KUKA KRL program: SCHUNK_GRASPINGKIT.src, SCHUNK_GRASPINGKIT.dat

--- SCHUNK_GRASPINGKIT.src ---
&ACCESS RVO4
&REL 37
&PARAM EDITMASK = *
&PARAM TEMPLATE = C:\KRC\Roboter\Template\ExpertVorgabe
&PARAM DISKPATH = KRC:\R1\Program\2DG
DEF SCHUNK_GRASPINGKIT( )
   INT v,s,c
   ;FOLD INI
      ;FOLD BASISTECH INI
         BAS (#INITMOV,0 )
      ;ENDFOLD (BASISTECH INI)
      ;FOLD USER INI
         ;Make your modifications here
      ;ENDFOLD (USER INI)
      ;ENDFOLD (INI)
   ;Example Program
   ;Init SVC
   SCHUNK_connect_SVC()
   v=SCHUNK_getVersion_SVC()
   ;If not v>=4 you need to update your device
   s=SCHUNK_getState_SVC()
   s=SCHUNK_getState_SVC()
   ;Add error handling if not s==2, meaning SVC is not operational
   SCHUNK_register_SVC()
   ;Init Robot and gripper
   ;Load the project that matches your application. Here project 14
   SCHUNK_setProject_SVC(14)
   ;Activate tool and workspace
   SCHUNK_setTool_SVC(1)
   SCHUNK_setWorkspace_SVC(1)
   ;Set grasp mode and object class according to your application
   SCHUNK_getGrasp_SVC(3,0,1)
   ;Different example with specified objectID=8 and graspMode=2
   ;SCHUNK_getGrasp_SVC(2,8,2)
   ;Check your edits in the $config.dat to see to which global variales the result was written
   ;Add your own error handling if replyCodeSCHUNK is not 1 meaning no part was grasped
   ;Activate your feeding system if candidateCountSCHUNK is too low
   ;Send Grasp Feedback (no effect in V4)
   SCHUNK_graspFeedback_SVC(0)
   ;Get count of all objects without planning a grasp
   c=SCHUNK_objectCount_SVC(1)
   ;with specified ObjectID
   ;c=SCHUNK_objectCount_SVC(8)
   ;Send robot pose (for robot calibration) Make sure robot position is in correct tool and base for this
   SCHUNK_robotCalib_SVC()
   ;Disconnect once finished
   SCHUNK_disconnect_SVC()
END
;FOLD SCHUNK 2D Grasping Kit Methods
   ;www.schunk.com/vision
   ;Includes methods to use the TCP/IP connection of the 2D Grasping Kit and use its commands
   ;This is not intended to move your robot, call this functions for your custom project
   ;Provided by: SCHUNK SE & Co. KG
   ;Author: Fabian Reinwald
   ;Created: 24.07.2023
   ;Last changed: 11.06.2025
   ;Keep in mind that this here needs a SCHUNK_2DGrasping.xml EthernetKRL configuration file
   ;<ETHERNETKRL>
   ;<CONFIGURATION>
      ;<EXTERNAL>
         ;<IP>172.31.1.76</IP>
         ;<PORT>42001</PORT>
         ;<TYPE>Server</TYPE>
      ;</EXTERNAL>
   ;</CONFIGURATION>
   ;<RECEIVE>
      ;<RAW>
         ;<ELEMENT Tag="SVCResponse" Type="BYTE" Set_Flag="12" SIZE="80" />
      ;</RAW>
   ;</RECEIVE>
   ;<SEND>
      ;<RAW>
         ;<ELEMENT Tag="SVCRequest" TYPE="BYTE" Set_Flag="13" SIZE="80"/>
      ;</RAW>
   ;</SEND>
   ;</ETHERNETKRL>
   ;File has to be stored at Config/User/Common/EthernetKRL/SCHUNK_2DGrasping.xml
   ;IP describes the IP adress that was set in the network settings of the SVC(SCHUNK Vision Controller)
   ;$Flag12 is used to show an incoming connection, change in xml file if needed and EKI_FLAG in .dat
   ;Tested with EthernetKRL 3.2.4
;ENDFOLD (SCHUNK 2D Grasping Kit Methods)
;Calling this function first is mandatory to establish a connection
GLOBAL DEF SCHUNK_connect_SVC()
   RET=EKI_Init("SCHUNK_2DGrasping")
   RET=EKI_Open("SCHUNK_2DGrasping")
END
;Returns the highest supported comm version by the SCHUNK Vision Controller
GLOBAL DEFFCT INT SCHUNK_getVersion_SVC()
   Prefix[]=SVC_prefix()
   Header[]=SVC_header(getVersionCode)
   Body[]=SVC_empty_body()
   OFFSET=0
   CAST_TO(Request[],OFFSET,Prefix[],Header[],Body[])
   RET = EKI_Send("SCHUNK_2DGrasping",Request[])
   FOR i=1 TO 80
      Response[i]=0
   ENDFOR
   WAIT FOR $FLAG[EKI_FLAG]
   RET=EKI_GetString("SCHUNK_2DGrasping","SVCResponse",Response[])
   $FLAG[EKI_FLAG]=FALSE
   OFFSET=10
   CAST_FROM(Response[],OFFSET,versionBuffer[])
   ;Buffers to variables
   versionSCHUNK=uint16_to_int(versionBuffer[])
   RETURN(versionSCHUNK)
ENDFCT
;Requests the current state of the SCHUNK Vision Controller.
;For state=/=2 you should probably code some exception handling as the device is not operational is that case
GLOBAL DEFFCT INT SCHUNK_getState_SVC()
   Prefix[]=SVC_prefix()
   Header[]=SVC_header(getStateCode)
   Body[]=SVC_empty_body()
   OFFSET=0
   CAST_TO(Request[],OFFSET,Prefix[],Header[],Body[])
   RET = EKI_Send("SCHUNK_2DGrasping",Request[])
   FOR i=1 TO 80
      Response[i]=0
   ENDFOR
   WAIT FOR $FLAG[EKI_FLAG]
   RET=EKI_GetString("SCHUNK_2DGrasping","SVCResponse",Response[])
   $FLAG[EKI_FLAG]=FALSE
   OFFSET=12
   CAST_FROM(Response[],OFFSET,stateBuffer[])
   stateSCHUNK=uint8_to_int(stateBuffer[])
   RETURN(stateSCHUNK)
ENDFCT
;This lets the SCHUNK Vision Controller know that it is connected to a KUKA Robot
;Calling this is the easiest way to check if your communication is working
GLOBAL DEF SCHUNK_register_SVC()
   Prefix[]=SVC_prefix()
   Header[]=SVC_header(registerClient)
   Body[]=SVC_register_client_body()
   OFFSET=0
   CAST_TO(Request[],OFFSET,Prefix[],Header[],Body[])
   RET = EKI_Send("SCHUNK_2DGrasping",Request[])
   FOR i=1 TO 80
      Response[i]=0
   ENDFOR
   WAIT FOR $FLAG[EKI_FLAG]
   RET=EKI_GetString("SCHUNK_2DGrasping","SVCResponse",Response[])
   $FLAG[EKI_FLAG]=FALSE
END
;Activates a project. The regarding ID can be seen in the web frontend
GLOBAL DEF SCHUNK_setProject_SVC(projectID:IN)
   INT projectID
   Prefix[]=SVC_prefix()
   Header[]=SVC_header(setProject)
   Body[]=SVC_set_project_body(projectID)
   OFFSET=0
   CAST_TO(Request[],OFFSET,Prefix[],Header[],Body[])
   RET = EKI_Send("SCHUNK_2DGrasping",Request[])
   FOR i=1 TO 80
      Response[i]=0
   ENDFOR
   WAIT FOR $FLAG[EKI_FLAG]
   RET=EKI_GetString("SCHUNK_2DGrasping","SVCResponse",Response[])
   $FLAG[EKI_FLAG]=FALSE
END
;Activates a tool. The regarding ID can be seen in the web frontend
GLOBAL DEF SCHUNK_setTool_SVC(toolID:IN)
   INT toolID
   Prefix[]=SVC_prefix()
   Header[]=SVC_header(setTool)
   Body[]=SVC_set_tool_body(toolID)
   OFFSET=0
   CAST_TO(Request[],OFFSET,Prefix[],Header[],Body[])
   RET = EKI_Send("SCHUNK_2DGrasping",Request[])
   FOR i=1 TO 80
      Response[i]=0
   ENDFOR
   WAIT FOR $FLAG[EKI_FLAG]
   RET=EKI_GetString("SCHUNK_2DGrasping","SVCResponse",Response[])
   $FLAG[EKI_FLAG]=FALSE
END
;Activates a workspace. The regarding ID can be seen in the web frontend
GLOBAL DEF SCHUNK_setWorkspace_SVC(workspaceID:IN)
   INT workspaceID
   Prefix[]=SVC_prefix()
   Header[]=SVC_header(setWorkspace)
   Body[]=SVC_set_workspace_body(workspaceID)
   OFFSET=0
   CAST_TO(Request[],OFFSET,Prefix[],Header[],Body[])
   RET = EKI_Send("SCHUNK_2DGrasping",Request[])
   FOR i=1 TO 80
      Response[i]=0
   ENDFOR
   WAIT FOR $FLAG[EKI_FLAG]
   RET=EKI_GetString("SCHUNK_2DGrasping","SVCResponse",Response[])
   $FLAG[EKI_FLAG]=FALSE
END
;This function requests a grasp pose. It is recommended to check if replyCodeSCHUNK==1,else there is no grasp
GLOBAL DEF SCHUNK_getGrasp_SVC(graspMode:IN, objectID:IN,selCriterion:IN)
   INT graspMode,objectID,selCriterion
   Prefix[]=SVC_prefix()
   Header[]=SVC_header(getGrasp)
   Body[]=SVC_get_grasp_body(graspMode, objectID, selCriterion)
   OFFSET=0
   CAST_TO(Request[],OFFSET,Prefix[],Header[],Body[])
   RET = EKI_Send("SCHUNK_2DGrasping",Request[])
   FOR i=1 TO 80
      Response[i]=0
   ENDFOR
   WAIT FOR $FLAG[EKI_FLAG]
   RET=EKI_GetString("SCHUNK_2DGrasping","SVCResponse",Response[])
   $FLAG[EKI_FLAG]=FALSE
   ;CAST_FROM is limited to 10 variables at once
   OFFSET=0
   CAST_FROM(Response[],OFFSET,preVersionBuffer[],lengthBuffer[],commTypeBuffer[],replyCodeBuffer[],replyCounterBuffer[],msgTypeBuffer[],graspModeBuffer[],objectIDBuffer[])
   OFFSET=16
   CAST_FROM(Response[],OFFSET,objectInstanceBuffer[],poseFormatBuffer[],referenceFrameBuffer[],strokeBuffer[],objectOffsetXBuffer[],objectOffsetYBuffer[],objectOffsetRZBuffer[])
   OFFSET=36
   CAST_FROM(Response[],OFFSET,centerOffsetXBuffer[],centerOffsetYBuffer[],graspPoseXBuffer[],graspPoseYBuffer[],graspPoseZBuffer[],graspPoseABuffer[],graspPoseBBuffer[],graspPoseCBuffer[])
   OFFSET=72
   CAST_FROM(Response[],OFFSET,candidateCountBuffer[],objectCountBuffer[])
   ;Buffers to variables
   preVersionSCHUNK=uint16_to_int(preVersionBuffer[])
   lengthSCHUNK=uint32_to_int(lengthBuffer[])
   commTypeSCHUNK=uint8_to_int(commTypeBuffer[])
   replyCodeSCHUNK=uint8_to_int(replyCodeBuffer[])
   replyCounterSCHUNK=uint8_to_int(replyCounterBuffer[])
   msgTypeSCHUNK=uint8_to_int(msgTypeBuffer[])
   graspModeSCHUNK=uint8_to_int(graspModeBuffer[])
   objectIDSCHUNK=uint16_to_int(objectIDBuffer[])
   objectInstanceSCHUNK=uint16_to_int(objectInstanceBuffer[])
   poseFormatSCHUNK=uint8_to_int(poseFormatBuffer[])
   referenceFrameSCHUNK=uint8_to_int(referenceFrameBuffer[])
   strokeSCHUNK=uint32_to_int(strokeBuffer[])
   objectOffsetXSCHUNK=uint32_to_int(objectOffsetXBuffer[])
   objectOffsetXSCHUNK=objectOffsetXSCHUNK/1000
   objectOffsetYSCHUNK=uint32_to_int(objectOffsetYBuffer[])
   objectOffsetYSCHUNK=objectOffsetYSCHUNK/1000
   objectOffsetRZSCHUNK=uint32_to_int(objectOffsetRZBuffer[])
   objectOffsetRZSCHUNK=objectOffsetRZSCHUNK/1000000
   xCenterOffsetSCHUNK=uint32_to_int(centerOffsetXBuffer[])
   xCenterOffsetSCHUNK=xCenterOffsetSCHUNK/1000
   yCenterOffsetSCHUNK=uint32_to_int(centerOffsetYBuffer[])
   yCenterOffsetSCHUNK=yCenterOffsetSCHUNK/1000
   poseXSCHUNK=uint32_to_int(graspPoseXBuffer[])
   poseXSCHUNK=poseXSCHUNK/1000
   poseYSCHUNK=uint32_to_int(graspPoseYBuffer[])
   poseYSCHUNK=poseYSCHUNK/1000
   poseZSCHUNK=uint32_to_int(graspPoseZBuffer[])
   poseZSCHUNK=poseZSCHUNK/1000
   poseASCHUNK=uint32_to_int(graspPoseABuffer[])
   poseASCHUNK=poseASCHUNK/1000000
   poseBSCHUNK=uint32_to_int(graspPoseBBuffer[])
   poseBSCHUNK=poseBSCHUNK/1000000
   poseCSCHUNK=uint32_to_int(graspPoseCBuffer[])
   poseCSCHUNK=poseCSCHUNK/1000000
   candidateCountSCHUNK=uint16_to_int(candidateCountBuffer[])
   objectCountSCHUNK=uint16_to_int(objectCountBuffer[])
END
;Function to report back to the SVC if a grasp was successfull. Has no effect on Version 3
GLOBAL DEF SCHUNK_graspFeedback_SVC(graspFeedback: in)
   INT graspFeedback
   Prefix[]=SVC_prefix()
   Header[]=SVC_header(graspFeedbackCode)
   Body[]=SVC_grasp_feedback_body(graspFeedback)
   OFFSET=0
   CAST_TO(Request[],OFFSET,Prefix[],Header[],Body[])
   RET = EKI_Send("SCHUNK_2DGrasping",Request[])
   FOR i=1 TO 80
      Response[i]=0
   ENDFOR
   WAIT FOR $FLAG[EKI_FLAG]
   RET=EKI_GetString("SCHUNK_2DGrasping","SVCResponse",Response[])
   $FLAG[EKI_FLAG]=FALSE
END
;Function to count detected objects in the scene. If objectClass=0 all classes are counted
GLOBAL DEFFCT INT SCHUNK_objectCount_SVC(objectClass: in)
   INT objectClass
   Prefix[]=SVC_prefix()
   Header[]=SVC_header(getObjectCount)
   Body[]=SVC_object_count_body(objectClass)
   OFFSET=0
   CAST_TO(Request[],OFFSET,Prefix[],Header[],Body[])
   RET = EKI_Send("SCHUNK_2DGrasping",Request[])
   FOR i=1 TO 80
      Response[i]=0
   ENDFOR
   WAIT FOR $FLAG[EKI_FLAG]
   RET=EKI_GetString("SCHUNK_2DGrasping","SVCResponse",Response[])
   $FLAG[EKI_FLAG]=FALSE
   OFFSET=72
   CAST_FROM(Response[],OFFSET,candidateCountBuffer[])
   OFFSET=74
   CAST_FROM(Response[],OFFSET,objectCountBuffer[])
   candidateCountSCHUNK=uint16_to_int(candidateCountBuffer[])
   objectCountSCHUNK=uint16_to_int(objectCountBuffer[])
   RETURN objectCountSCHUNK
ENDFCT
;Function for calibration method with board mounted to flange or camera on robot
GLOBAL DEF SCHUNK_robotCalib_SVC()
   Prefix[]=SVC_prefix()
   Header[]=SVC_header(robotPose)
   Body[]=SVC_robot_pose($POS_ACT.X,$POS_ACT.Y,$POS_ACT.Z,$POS_ACT.A*1000,$POS_ACT.B*1000,$POS_ACT.C*1000)
   OFFSET=0
   CAST_TO(Request[],OFFSET,Prefix[],Header[],Body[])
   RET = EKI_Send("SCHUNK_2DGrasping",Request[])
   FOR i=1 TO 80
      Response[i]=0
   ENDFOR
   WAIT FOR $FLAG[EKI_FLAG]
   RET=EKI_GetString("SCHUNK_2DGrasping","SVCResponse",Response[])
   $FLAG[EKI_FLAG]=FALSE
END
;Clear your communication and disconnect from the SCHUNK Vision Controller
GLOBAL DEF SCHUNK_disconnect_SVC()
   RET=EKI_Close("SCHUNK_2DGrasping")
   RET=EKI_Clear("SCHUNK_2DGrasping")
END
;----------------------------HELPERS-------------------------------------------
DEFFCT CHAR[6] SVC_prefix()
   CHAR prefix[6], readVersionBuffer[4]
   FOR i=1 TO 6
      prefix[i]=0
   ENDFOR
   OFFSET=0
   CAST_TO(readVersionBuffer[],OFFSET,version)
   OFFSET=0
   CAST_TO(lengthBuffer[],OFFSET,length)
   OFFSET=0
   CAST_TO(prefix[],OFFSET,readVersionBuffer[2],readVersionBuffer[1],lengthBuffer[4],lengthBuffer[3],lengthBuffer[2],lengthBuffer[1])
   RETURN prefix[]
ENDFCT
DEFFCT CHAR[4] SVC_header(msgType:IN)
   INT msgType
   CHAR header[4],readCommTypeBuffer[4],readReplyCodeBuffer[4],readReplyCounterBuffer[4],readMsgTypeBuffer[4]
   FOR i=1 TO 4
      header[i]=0
   ENDFOR
   OFFSET=0
   CAST_TO(readCommTypeBuffer[],OFFSET,commType)
   OFFSET=0
   CAST_TO(readReplyCodeBuffer[],OFFSET,replyCode)
   OFFSET=0
   CAST_TO(readReplyCounterBuffer[],OFFSET,replyCounter)
   OFFSET=0
   CAST_TO(readMsgTypeBuffer[],OFFSET,msgType)
   OFFSET=0
   CAST_TO(header[],OFFSET,readCommTypeBuffer[1],readReplyCodeBuffer[1],readReplyCounterBuffer[1],readMsgTypeBuffer[1])
   RETURN header[]
ENDFCT
DEFFCT CHAR[70] SVC_empty_body()
   CHAR body[70]
   FOR i=1 TO 70
      body[i]=0
   ENDFOR
   RETURN body[]
ENDFCT
DEFFCT CHAR[70] SVC_register_client_body()
   CHAR body[70],readClientBuffer[4]
   FOR i=1 TO 70
      body[i]=0
   ENDFOR
   OFFSET=0
   CAST_TO(readClientBuffer[],OFFSET,client)
   OFFSET=0
   CAST_TO(body[],OFFSET,readClientBuffer[1])
   RETURN body[]
ENDFCT
DEFFCT CHAR[70] SVC_set_project_body(projectID:IN)
   INT projectID
   CHAR body[70]
   FOR i=1 TO 70
      body[i]=0
   ENDFOR
   OFFSET=0
   CAST_TO(projectIDBuffer[],OFFSET,projectID)
   OFFSET=8
   CAST_TO(body[],OFFSET,projectIDBuffer[2],projectIDBuffer[1])
   RETURN body[]
ENDFCT
DEFFCT CHAR[70] SVC_set_tool_body(toolID:IN)
   INT toolID
   CHAR body[70]
   FOR i=1 TO 70
      body[i]=0
   ENDFOR
   OFFSET=0
   CAST_TO(toolIDBuffer[],OFFSET,toolID)
   OFFSET=10
   CAST_TO(body[],OFFSET,toolIDBuffer[2],toolIDBuffer[1])
   RETURN body[]
ENDFCT
DEFFCT CHAR[70] SVC_set_workspace_body(workspaceID:IN)
   INT workspaceID
   CHAR body[70]
   FOR i=1 TO 70
      body[i]=0
   ENDFOR
   OFFSET=0
   CAST_TO(workspaceIDBuffer[],OFFSET,workspaceID)
   OFFSET=12
   CAST_TO(body[],OFFSET,workspaceIDBuffer[2],workspaceIDBuffer[1])
   RETURN body[]
ENDFCT
DEFFCT CHAR[70] SVC_get_grasp_body(graspMode:IN,objectID:IN,selCriterion:IN)
   INT graspMode,objectID,selCriterion
   CHAR body[70],readGraspModeBuffer[4],readObjectIDBuffer[4],readselCriterionBuffer[4],readPoseFormatBuffer[4]
   FOR i=1 TO 70
      body[i]=0
   ENDFOR
   OFFSET=0
   CAST_TO(readGraspModeBuffer[],OFFSET,graspMode)
   OFFSET=0
   CAST_TO(readObjectIDBuffer[],OFFSET,objectID)
   OFFSET=0
   CAST_TO(readselCriterionBuffer[],OFFSET,selCriterion)
   OFFSET=0
   CAST_TO(readPoseFormatBuffer[],OFFSET,poseFormat)
   OFFSET=1
   CAST_TO(body[],OFFSET,readGraspModeBuffer[1],readObjectIDBuffer[2],readObjectIDBuffer[1],readselCriterionBuffer[1],readPoseFormatBuffer[1])
   RETURN body[]
ENDFCT
DEFFCT CHAR[70] SVC_grasp_feedback_body(feedback:IN)
   INT feedback
   CHAR body[70],readGraspFeedbackBuffer[4]
   FOR i=1 TO 70
      body[i]=0
   ENDFOR
   OFFSET=0
   CAST_TO(readGraspFeedbackBuffer[],OFFSET,feedback)
   OFFSET=6
   CAST_TO(body[],OFFSET,readGraspFeedbackBuffer[1])
   RETURN body[]
ENDFCT
DEFFCT CHAR[70] SVC_object_count_body(objectClass:IN)
   INT objectClass
   CHAR body[70], readobjectIDBuffer[4]
   FOR i=1 TO 70
      body[i]=0
   ENDFOR
   OFFSET=0
   CAST_TO(readobjectIDBuffer[],OFFSET,objectClass)
   OFFSET=2
   CAST_TO(body[],OFFSET,readobjectIDBuffer[2],readobjectIDBuffer[1])
   RETURN body[]
ENDFCT
DEFFCT CHAR[70] SVC_robot_pose(X:IN,Y:IN,Z:IN,A:IN,B:IN,C:IN)
   CHAR body[70],readPoseFormatBuffer[4]
   REAL X,Y,Z,A,B,C
   CHAR Xchar[4],Ychar[4],Zchar[4],Achar[4],Bchar[4],Cchar[4]
   FOR i=1 TO 70
      body[i]=0
   ENDFOR
   OFFSET=0
   CAST_TO(readPoseFormatBuffer[],OFFSET,poseFormat)
   OFFSET=1
   CAST_TO(body[],OFFSET,FALSE,FALSE,FALSE,FALSE,readPoseFormatBuffer[1])
   Xchar[]=real_to_kilo_int_char(X)
   Ychar[]=real_to_kilo_int_char(Y)
   Zchar[]=real_to_kilo_int_char(Z)
   Achar[]=real_to_kilo_int_char(A)
   Bchar[]=real_to_kilo_int_char(B)
   Cchar[]=real_to_kilo_int_char(C)
   OFFSET=14
   CAST_TO(body[],OFFSET,Xchar[],Ychar[],Zchar[],Achar[],Bchar[],Cchar[])
   RETURN body[]
ENDFCT
;Takes a REAL as input (for example from $POS_ACT, converts it to array of int values)
;multiplies with 1000 for microunit and changes to Big-Endian
DEFFCT CHAR[4] real_to_kilo_int_char(f:IN)
   DECL REAL f
   DECL INT i
   DECL CHAR buf[4], resp[4]
   OFFSET=0
   f=f*1000
   i=f
   OFFSET=0
   CAST_TO(buf[],OFFSET,i)
   OFFSET=0
   CAST_TO(resp[],OFFSET,buf[4],buf[3],buf[2],buf[1])
   RETURN resp[]
ENDFCT
DEFFCT INT uint8_to_int(uint8Buffer[]:IN)
   CHAR uint8Buffer[]
   INT i
   OFFSET=0
   CAST_TO(intConverter[],OFFSET,uint8Buffer[1],FALSE,FALSE,FALSE)
   OFFSET=0
   CAST_FROM(intConverter[],OFFSET,i)
   RETURN i
ENDFCT
DEFFCT INT uint16_to_int(uint16Buffer[]:IN)
   CHAR uint16Buffer[]
   INT i
   OFFSET=0
   CAST_TO(intConverter[],OFFSET,uint16Buffer[2],uint16Buffer[1],FALSE,FALSE)
   OFFSET=0
   CAST_FROM(intConverter[],OFFSET,i)
   RETURN i
ENDFCT
DEFFCT INT uint32_to_int(uint32Buffer[]:IN)
   CHAR uint32Buffer[]
   INT i
   OFFSET=0
   CAST_TO(intConverter[],OFFSET,uint32Buffer[4],uint32Buffer[3],uint32Buffer[2],uint32Buffer[1])
   OFFSET=0
   CAST_FROM(intConverter[],OFFSET,i)
   RETURN i
ENDFCT

--- SCHUNK_GRASPINGKIT.dat ---
&ACCESS RVO1
&REL 49
&PARAM EDITMASK = *
&PARAM TEMPLATE = C:\KRC\Roboter\Template\ExpertVorgabe
&PARAM DISKPATH = KRC:\R1\Program\2DG
DEFDAT  SCHUNK_GRASPINGKIT PUBLIC
;www.schunk.com/vision
;Keep KUKA Byte swap in mind. If SVC needs a 'H12345678' you would create a 'H78563412' in KUKA
;-----------------------------------------------------------------------------------------
;Prefix
DECL CONST INT version=4
DECL CHAR preVersionBuffer[2]
DECL CHAR versionBuffer[2]
DECL CONST INT length=74 ; we send fixed length of total 80. Header=6 so baseLength=80-6=74
DECL CHAR lengthBuffer[4]
;Header
DECL CONST INT commType=1
DECL CHAR commTypeBuffer[1]
DECL CONST INT replyCode=0
DECL CHAR replyCodeBuffer[1]
DECL CONST INT replyCounter=0
DECL CHAR replyCounterBuffer[1]
;Header Message Types
DECL INT msgType
DECL CONST INT getVersionCode=1
DECL CONST INT getStateCode=2
DECL CONST INT registerClient=3
DECL CONST INT setProject=4
DECL CONST INT setTool=5
DECL CONST INT setWorkspace=6
DECL CONST INT getGrasp=16
DECL CONST INT graspFeedbackCode=17
DECL CONST INT getObjectCount=32
DECL CONST INT robotPose=48
DECL CHAR msgTypeBuffer[1]
;Request-Body
DECL CONST INT client=2 ;Set in registerClient request function
DECL INT graspMode ;Set in getGrasp request function
DECL CHAR graspModeBuffer[4]
DECL INT objectID ;Set in getGrasp request function
DECL CHAR objectIDBuffer[4]
DECL INT selCriterion ;Set in getGrasp request function
DECL CONST INT poseFormat=17
DECL CHAR poseFormatBuffer[1]
DECL INT feedback ;Not yet supported with V4
DECL INT projectID ;Set in setProject request function
DECL CHAR projectIDBuffer[4]
DECL INT toolID ;Set in setTool request function
DECL CHAR toolIDBuffer[4]
DECL INT workspaceID ;Set in setWorkspace request function
DECL CHAR workspaceIDBuffer[4]
;Response Buffer - values will be stored in global config.dat variables
DECL CHAR stateBuffer[1]
DECL CHAR objectInstanceBuffer[2]
DECL CHAR referenceFrameBuffer[1]
DECL CHAR strokeBuffer[4]
DECL CHAR objectOffsetXBuffer[4]
DECL CHAR objectOffsetYBuffer[4]
DECL CHAR objectOffsetRZBuffer[4]
DECL CHAR centerOffsetXBuffer[4]
DECL CHAR centerOffsetYBuffer[4]
DECL CHAR graspPoseXBuffer[4]
DECL CHAR graspPoseYBuffer[4]
DECL CHAR graspPoseZBuffer[4]
DECL CHAR graspPoseABuffer[4]
DECL CHAR graspPoseBBuffer[4]
DECL CHAR graspPoseCBuffer[4]
DECL CHAR candidateCountBuffer[2]
DECL CHAR objectCountBuffer[2]
;Paste the following into your config.dat
;====================================
; Userdefined Variables for SCHUNK 2DGK
;====================================
;INT preVersionSCHUNK
;INT lengthSCHUNK
;
;INT commTypeSCHUNK
;INT replyCodeSCHUNK
;INT replyCounterSCHUNK
;INT msgTypeSCHUNK
;
;INT versionSCHUNK
;INT stateSCHUNK
;
;INT graspModeSCHUNK
;INT objectIDSCHUNK
;INT objectInstanceSCHUNK
;INT strokeSCHUNK;[micrometers] SCHUNK Grippers take this as Input
;REAL angleOffsetSCHUNK;[degrees]
;REAL xCenterOffsetSCHUNK;[millimeters]
;REAL yCenterOffsetSCHUNK;[millimeters]
;REAL zCenteroffsetSCHUNK;[millimeters]
;INT toolSCHUNK
;INT poseFormatSCHUNK
;INT referenceFrameSCHUNK
;INT objectOffsetXSCHUNK
;INT objectOffsetYSCHUNK
;INT objectOffsetRZSCHUNK
;
;REAL poseXSCHUNK;[millimeters]
;REAL poseYSCHUNK;[millimeters]
;REAL poseZSCHUNK;[millimeters]
;
;REAL poseASCHUNK;[degrees]
;REAL poseBSCHUNK;[degrees]
;REAL poseCSCHUNK;[degrees]
;
;INT objectCountSCHUNK
;INT candidateCountSCHUNK
;----------------------------------------------------------------------------------------
DECL EKI_STATUS RET
DECL CONST INT EKI_FLAG=12 ;
DECL CHAR Prefix[6]
DECL CHAR Header[4]
DECL CHAR Body[70]
DECL CHAR Request[80]
DECL CHAR Response[80]
DECL INT i
DECL INT OFFSET=4

DECL CHAR intConverter[4]
ENDDAT
